// Mitsubishi GX Works2 project: LRI - PLC - SEMARO FUN BLOC   PLC: Q03UDV

// task Task_01 (event TRUE, interval 0, priority 31): POU_01

PROGRAM POU_01
VAR
  CTU_1 : CTU;
  CTD_1 : CTD;
  CTUD_1 : CTUD;
  CTUD_CTUD_11 : CTUD;
END_VAR
(* structured ladder/FBD written out as ST: instructions are called as NAME(EN, inputs, outputs); _pN, _eN, _tN stand for wires *)
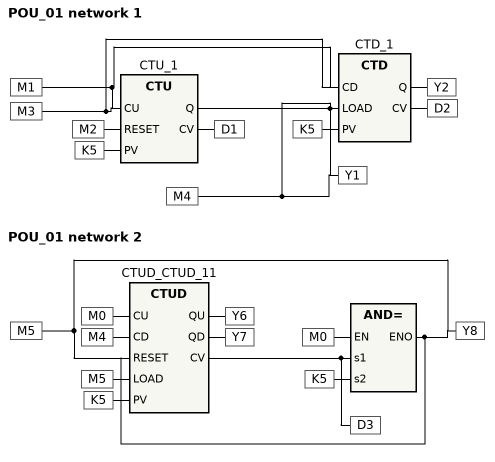
(* network 1 *)
_p1 := M1 OR M3;
CTU_1(CU := _p1, RESET := M2, PV := K5, CV => D1);
_p2 := CTU_1.Q OR M4;
Y1 := _p2;
CTD_1(CD := _p1, LOAD := _p2, PV := K5, Q => Y2, CV => D2);
(* network 2 *)
_e1 := AND=(M0, CTUD_CTUD_11.CV, K5);
_p2 := M5 OR _e1;
CTUD_CTUD_11(CU := M0, CD := M4, RESET := _p2, LOAD := M5, PV := K5, QU => Y6, QD => Y7);
D3 := CTUD_CTUD_11.CV;
Y8 := _p2;
END_PROGRAM
